(* IEC 61131-3 sources: RL_MAR/experiments/comparison/llm4plc/results/gpt-4o-mini_20260506_100619/20260506_101912, 2 files *)

(* ---- generated_code_iteration_0.st ---- *)
ructured-text
START_ST
FUNCTION_BLOCK FB_SimpleCalculation
VAR_INPUT
    INPUT_VAR1 : INT := 2;
    VAR2 : INT := 0;
END_VAR

VAR_OUTPUT
    OUTPUT_VAR1 : INT;
    OUTPUT_VAR2 : INT;
END_VAR

VAR
    state : INT; // THE STATE VARIABLE
    COUNTER1 : INT := 0; // COUNTER FOR MULTIPLICATION
    COUNTER2 : INT := 0; // COUNTER FOR INCREMENTING
END_VAR

// Initialization
state := 0;
OUTPUT_VAR1 := 0;
OUTPUT_VAR2 := 0;

WHILE state <> 3 DO
    CASE state OF
        0: // STATE 0: INITIALIZE
            OUTPUT_VAR1 := 0;
            OUTPUT_VAR2 := 0;
            state := 1; // Move to multiplication state

        1: // STATE 1: MULTIPLY OUTPUT_VAR1
            IF COUNTER1 < 5 THEN
                OUTPUT_VAR1 := INPUT_VAR1 * (2 ** COUNTER1);
                COUNTER1 := COUNTER1 + 1; // Increment multiplication counter
            ELSE
                state := 2; // Move to increment state
            END_IF;

        2: // STATE 2: INCREMENT OUTPUT_VAR2
            IF COUNTER2 < 5 THEN
                OUTPUT_VAR2 := COUNTER2;
                COUNTER2 := COUNTER2 + 1; // Increment increment counter
            ELSE
                state := 3; // Move to finalize state
            END_IF;

        3: // STATE 3: FINALIZE
            // Final state, outputs are ready
            // No further actions required
    END_CASE;
END_WHILE;

END_FUNCTION_BLOCK
END_ST

(* ---- generated_code_iteration_1.st ---- *)
START_REASON
The errors in the original structured text (ST) code occurred because the exponentiation operator `**` is not valid in the context of the CODESYS environment, which requires the use of the multiplication operator `*` instead. The feedback specifically indicated that `**` should be replaced with `*`, which is a common requirement in many programming environments. Additionally, there were issues with the variable section closure, which should use `END_VAR` instead of `END_VAR_OUTPUT` or `END_VAR_INPUT`.

Given these points, I will correct the exponentiation operation and ensure the variable sections are properly closed.

END_REASON

START_ST
FUNCTION_BLOCK FB_SimpleCalculation
VAR_INPUT
    INPUT_VAR1 : INT := 2;
    VAR2 : INT := 0;
END_VAR

VAR_OUTPUT
    OUTPUT_VAR1 : INT;
    OUTPUT_VAR2 : INT;
END_VAR

VAR
    state : INT; // THE STATE VARIABLE
    COUNTER1 : INT := 0; // COUNTER FOR MULTIPLICATION
    COUNTER2 : INT := 0; // COUNTER FOR INCREMENTING
END_VAR

// Initialization
state := 0;
OUTPUT_VAR1 := 0;
OUTPUT_VAR2 := 0;

WHILE state <> 3 DO
    CASE state OF
        0: // STATE 0: INITIALIZE
            OUTPUT_VAR1 := 0;
            OUTPUT_VAR2 := 0;
            state := 1; // Move to multiplication state

        1: // STATE 1: MULTIPLY OUTPUT_VAR1
            IF COUNTER1 < 5 THEN
                OUTPUT_VAR1 := INPUT_VAR1 * (2 * COUNTER1); // Replace exponentiation with multiplication
                COUNTER1 := COUNTER1 + 1; // Increment multiplication counter
            ELSE
                state := 2; // Move to increment state
            END_IF;

        2: // STATE 2: INCREMENT OUTPUT_VAR2
            IF COUNTER2 < 5 THEN
                OUTPUT_VAR2 := COUNTER2;
                COUNTER2 := COUNTER2 + 1; // Increment increment counter
            ELSE
                state := 3; // Move to finalize state
            END_IF;

        3: // STATE 3: FINALIZE
            // Final state, outputs are ready
            // No further actions required
    END_CASE;
END_WHILE;

END_FUNCTION_BLOCK
END_ST
